TYPE (* DataPanel Modules with medium IO density AQ Struct *)
  (* Version 1.0, 2026-01-16, generated *)
  PACKAGE DataPanel::io::MI::AQ;
  DataPanel_MI_AQ_S : STRUCT
    Pin : USINT := 255;
  END_STRUCT;
END_TYPE
